// TIA Portal V19 export
TYPE "IPC_Msg_Log_PPRF"
   STRUCT
      Id : DInt;   // Identificativo progressivo univoco del messaggio (0 = cella vuota)
      timestamp : String;   // Timestamp evento formato ISO: YYYY-MM-DD HH:MM:SS.mmm
      topic : UDInt;   // Numero del programma profilo
      payLoad_01 : String;   // Record di valori [P001]=Value; .... [P015]=Valore
      payLoad_02 : String;   // [P016]..P[030]
      payLoad_03 : String;   // [P031]..P[045]
      payLoad_04 : String;   // [P046]..P[060]
      payLoad_05 : String;   // [P061]..P[075]
      payLoad_06 : String;   // [P076]..P[090]
      payLoad_07 : String;   // [P091]..P[105]
      payLoad_08 : String;   // [P106]..P[120]
      payLoad_09 : String;   // [P121]..P[135]
      payLoad_10 : String;   // [P136]..P[150]
      payLoad_11 : String;   // [P153]..P[157]
      payLoad_12 : String;   // Libero per opzioni future
      payLoad_13 : String;   // Libero per opzioni future
      payLoad_14 : String;   // Libero per opzioni future
      payLoad_15 : String;   // Libero per opzioni future
      payLoad_16 : String;   // Libero per opzioni future
   END_STRUCT;
END_TYPE
